// Mitsubishi GX Works2 project: 고속 타이머   PLC: Q02/Q02H

PROGRAM MAIN
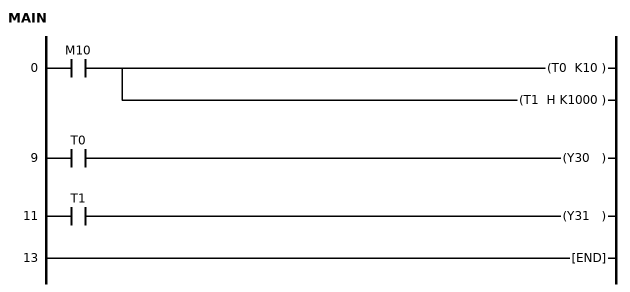
0     LD      M10
      OUT     T0 K10
      OUTH    T1 K1000
9     LD      T0
      OUT     Y30
11    LD      T1
      OUT     Y31
13    END
END_PROGRAM
